Fanuc KAREL source: compact_preamble.KL

PROGRAM KB00184
%NOLOCKGROUP
VAR
P1 : STRING[80];P2:INTEGER;P3:INTEGER;P4:INTEGER
BEGIN
P1='A'
P2=1
P3=1
P4=1
SET_TSK_ATTR(P1,P2,P3,P4)
END KB00184
